FUNCTION accum : BOOL
VAR_IN_OUT
	a,b:ARRAY[*,*] OF LREAL;
END_VAR
VAR_INPUT
	m,n:SINT;
END_VAR
VAR
	i,j:SINT;
END_VAR

		
FOR i:=0 TO m-1 DO
        FOR j:=0  TO n-1 DO 
            a[i,j] := a[i,j]+b[i,j];
			END_FOR
	END_FOR
	accum:=true;

END_FUNCTION

(* stored: Version 1.1.0.1, ProductVersion 3.1.4024.12
   POU accum: Id {a0ed3e46-6bcf-493a-aa32-9b22363e96f1}, SpecialFunc None *)
